DATA_BLOCK "DB_HardwareDataTypes"
{ S7_Optimized_Access := 'TRUE' }
VERSION : 0.1
NON_RETAIN
   VAR
      AOM_IDENT_0x1 : AOM_IDENT;   // AOM_IDENT: Testvalue 1
      CONN_ANY_0x2 : CONN_ANY;   // CONN_ANY: Testvalue 1
      CONN_OUC_0x3 : CONN_OUC;   // CONN_OUC: Testvalue 1
      CONN_PRG_0x4 : CONN_PRG;   // CONN_PRG: Testvalue 1
      CONN_R_ID_0x5 : CONN_R_ID;   // CONN_R_ID: Testvalue 1
      DB_ANY_1001 : DB_ANY;   // DB_ANY: Testvalue 1
      DB_DYN_1002 : DB_DYN;   // DB_DYN: Testvalue 1
      DB_WWW_1003 : DB_WWW;   // DB_WWW: Testvalue 1
      EVENT_ANY_0x6 : EVENT_ANY;   // EVENT_ANY: Testvalue 1
      EVENT_ATT_0x7 : EVENT_ATT;   // EVENT_ATT: Testvalue 1
      EVENT_HWINT_0x8 : EVENT_HWINT;   // EVENT_HWINT: Testvalue 1
      HW_ANY_1004 : HW_ANY;   // HW_ANY: Testvalue 1
      HW_DEVICE_1005 : HW_DEVICE;   // HW_DEVICE: Testvalue 1
      HW_DPMASTER_1006 : HW_DPMASTER;   // HW_DPMASTER: Testvalue 1
      HW_DPSLAVE_1007 : HW_DPSLAVE;   // HW_DPSLAVE: Testvalue 1
      HW_HSC_1008 : HW_HSC;   // HW_HSC: Testvalue 1
      HW_IEPORT_1009 : HW_IEPORT;   // HW_IEPORT: Testvalue 1
      HW_INTERFACE_1010 : HW_INTERFACE;   // HW_INTERFACE: Testvalue 1
      HW_IO_1011 : HW_IO;   // HW_IO: Testvalue 1
      HW_IOSYSTEM_1012 : HW_IOSYSTEM;   // HW_IOSYSTEM: Testvalue 1
      HW_MODULE_1013 : HW_MODULE;   // HW_MODULE: Testvalue 1
      HW_PTO_1014 : HW_PTO;   // HW_PTO: Testvalue 1
      HW_PWM_1015 : HW_PWM;   // HW_PWM: Testvalue 1
      HW_SUBMODULE_1016 : HW_SUBMODULE;   // HW_SUBMODULE: Testvalue 1
      OB_ANY_1017 : OB_ANY;   // OB_ANY: Testvalue 1
      OB_ATT_1018 : OB_ATT;   // OB_ATT: Testvalue 1
      OB_CYCLIC_1019 : OB_CYCLIC;   // OB_CYCLIC: Testvalue 1
      OB_DELAY_1020 : OB_DELAY;   // OB_DELAY: Testvalue 1
      OB_DIAG_1021 : OB_DIAG;   // OB_DIAG: Testvalue 1
      OB_HWINT_1022 : OB_HWINT;   // OB_HWINT: Testvalue 1
      OB_PCYCLE_1023 : OB_PCYCLE;   // OB_PCYCLE: Testvalue 1
      OB_STARTUP_1024 : OB_STARTUP;   // OB_STARTUP: Testvalue 1
      OB_TIMEERROR_1025 : OB_TIMEERROR;   // OB_TIMEERROR: Testvalue 1
      OB_TOD_1026 : OB_TOD;   // OB_TOD: Testvalue 1
      PIP_1027 : PIP;   // PIP: Testvalue 1
      PORT_1028 : PORT;   // PORT: Testvalue 1
      RTM_1029 : RTM;   // RTM: Testvalue 1
   END_VAR


BEGIN
   AOM_IDENT_0x1 := 16#0001;
   CONN_ANY_0x2 := 16#0002;
   CONN_OUC_0x3 := 16#0003;
   CONN_PRG_0x4 := 16#0004;
   CONN_R_ID_0x5 := 16#0005;
   DB_ANY_1001 := 1001;
   DB_DYN_1002 := 1002;
   DB_WWW_1003 := 1003;
   EVENT_ANY_0x6 := 16#0006;
   EVENT_ATT_0x7 := 16#0007;
   EVENT_HWINT_0x8 := 16#0008;
   HW_ANY_1004 := 1004;
   HW_DEVICE_1005 := 1005;
   HW_DPMASTER_1006 := 1006;
   HW_DPSLAVE_1007 := 1007;
   HW_HSC_1008 := 1008;
   HW_IEPORT_1009 := 1009;
   HW_INTERFACE_1010 := 1010;
   HW_IO_1011 := 1011;
   HW_IOSYSTEM_1012 := 1012;
   HW_MODULE_1013 := 1013;
   HW_PTO_1014 := 1014;
   HW_PWM_1015 := 1015;
   HW_SUBMODULE_1016 := 1016;
   OB_ANY_1017 := 1017;
   OB_ATT_1018 := 1018;
   OB_CYCLIC_1019 := 1019;
   OB_DELAY_1020 := 1020;
   OB_DIAG_1021 := 1021;
   OB_HWINT_1022 := 1022;
   OB_PCYCLE_1023 := 1023;
   OB_STARTUP_1024 := 1024;
   OB_TIMEERROR_1025 := 1025;
   OB_TOD_1026 := 1026;
   PIP_1027 := 1027;
   PORT_1028 := 1028;
   RTM_1029 := 1029;

END_DATA_BLOCK

